PROGRAM MAIN
VAR
END_VAR

END_PROGRAM

(* stored: Version 1.1.0.1, ProductVersion 3.1.4024.5
   POU MAIN: Id {e32b1aa3-a44f-4c6b-8682-15ba4b138c6b}, SpecialFunc None *)
